// TIA Portal project "Project1" (V15.1)

(* hardware
DEVICE "ET 200SP station_2"  ET 200SP-Station
   slot 0: "Rack_0"  Rack  6ES5 710-8MAx1
   slot 1: "PLC_1"  CPU 1512SP F-1 PN  6ES7 512-1SK01-0AB0  V2.6
   slot 2: "DI 8x24VDC HF_1"  DI 8x24VDC HF  6ES7 131-6BF00-0CA0  V2.0
      slot 1: "DI 8x24VDC HF_1"  DI 8x24VDC HF
   slot 3: "DI 8x24VDC HF_2"  DI 8x24VDC HF  6ES7 131-6BF00-0CA0  V2.0
      slot 1: "DI 8x24VDC HF_2"  DI 8x24VDC HF
   slot 4: "DQ 8x24VDC/0.5A HF_1"  DQ 8x24VDC/0.5A HF  6ES7 132-6BF00-0CA0  V2.0
      slot 1: "DQ 8x24VDC/0.5A HF_1"  DQ 8x24VDC/0.5A HF
   slot 5: "DQ 8x24VDC/0.5A HF_2"  DQ 8x24VDC/0.5A HF  6ES7 132-6BF00-0CA0  V2.0
      slot 1: "DQ 8x24VDC/0.5A HF_2"  DQ 8x24VDC/0.5A HF
   slot 6: "CM 4xIO-Link_1"  CM 4xIO-Link  6ES7 137-6BD00-0BA0  V2.2
      slot 1: "CM 4xIO-Link_1"  6ES7 137-6BD00-0BA0
   slot 7: "Server module_1"  Server module  6ES7 193-6PA00-0AA0  V1.1
      slot 1: "Server module_1"  Server module
   slot 127: "BA 2xRJ45"  BA 2xRJ45  6ES7 193-6AR00-0AA0  V0.0
      slot 32769: "Port_1"  6ES7 193-6AR00-0AA0
      slot 32770: "Port_2"  6ES7 193-6AR00-0AA0
*)

// ===== PLC "PLC_1"  CPU 1512SP F-1 PN =====

VAR_GLOBAL   // PLC tag table "Conv_tag table"
   "start_btn" AT %I1.0 : Bool;
   "stop_btn" AT %I1.1 : Bool;
   "select_op_mode" AT %I1.2 : Bool;
   "reset_btn" AT %I1.3 : Bool;
   "carr_det_stop_pos" AT %I1.4 : Bool;
   "EM_stop" AT %I1.5 : Bool;
   "carr_det_conv_entry" AT %I1.6 : Bool;
   "carr_det_conv_exit" AT %I1.7 : Bool;
   "Carr_id_bit0_det" AT %I42.0 : Bool;
   "Carr_id_bit1_det" AT %I42.1 : Bool;
   "Carr_id_bit2_det" AT %I42.2 : Bool;
   "Carr_id_bit3_det" AT %I42.3 : Bool;
   "SW_s1" AT %I42.4 : Bool;
   "SW_s2" AT %I42.5 : Bool;
   "stop_cyl_low_end" AT %I42.7 : Bool;
   "SW_start_light" AT %Q1.0 : Bool;
   "SW_reset_light" AT %Q1.1 : Bool;
   "SW_func_Q1_light" AT %Q1.2 : Bool;
   "SW_func_Q2_light" AT %Q1.3 : Bool;
   "belt_forward" AT %Q1.4 : Bool;
   "belt_reverse" AT %Q1.5 : Bool;
   "select_belt_speed" AT %Q1.6 : Bool;
   "stop_cyl_mov_down" AT %Q1.7 : Bool;
   "coupling_signal_left" AT %Q42.4 : Bool;
   "coupling_signal_right" AT %Q42.5 : Bool;
END_VAR

DATA_BLOCK "idbAksjoner"   // DB1
{ S7_Optimized_Access := 'TRUE' }
VERSION : 0.1
// stored: InstanceOfName fbAksjoner
"fbAksjoner"
BEGIN
END_DATA_BLOCK

FUNCTION_BLOCK "fbAksjoner"   // FB1, SCL
{ S7_Optimized_Access := 'TRUE' }
VERSION : 0.1
   VAR_INPUT
      bStartBtn : Bool;
   END_VAR
   VAR_OUTPUT
      bStartBtnLight : Bool;
      bConveyerBeltForw : Bool;
   END_VAR
BEGIN
   IF #bStartBtn THEN
       #bStartBtnLight := true;
       #bConveyerBeltForw := true;
   ELSE
       #bStartBtnLight := FALSE;
       #bConveyerBeltForw := FALSE;
   END_IF;
END_FUNCTION_BLOCK

ORGANIZATION_BLOCK "Main"   // OB1, SCL, ProgramCycle
TITLE = "Main Program Sweep (Cycle)"
{ S7_Optimized_Access := 'TRUE' }
VERSION : 0.1
   VAR_INPUT
      Initial_Call : Bool;   // Initial call of this OB
      Remanence : Bool;   // =True, if remanent data are available
   END_VAR
BEGIN
   "idbAksjoner".bStartBtn := "start_btn";
   "idbAksjoner".bStartBtnLight := "SW_start_light";
   "idbAksjoner".bConveyerBeltForw := "belt_forward";

   "idbAksjoner"();
END_ORGANIZATION_BLOCK